FUNCTION "GestConsensoReal" : Void
{ S7_Optimized_Access := 'TRUE' }
VERSION : 0.1
   VAR_INPUT
      K_SegnaleMacchina : Int;
      K_Consenso : Int;
      K_TipoSendReceive : Int;   // Indica se è un segnale send o recive
      SegnaleIn : Real;   // Segnale in ingresso al blocco da inviare o ricevuto
   END_VAR

   VAR_OUTPUT
      OutSegnale : Real;
   END_VAR

   VAR_TEMP
      SegnaleForzatoOn : Bool;
      SegnaleForzatoOff : Bool;
      AbilitaTimeoutForzature : Bool;
      TimeoutForzature : Bool;
      ResettaForzature : Bool;
      PreOutSegnale : Real;
      StatoHmi : Int;
   END_VAR


BEGIN
	REGION Gestione delle forzature ad Hmi
	    #SegnaleForzatoOn := "SegnaliMacchina".S[#K_SegnaleMacchina].SR[#K_TipoSendReceive]."Real"[#K_Consenso].Hmi.ForzaturaOn;
	    #SegnaleForzatoOff := "SegnaliMacchina".S[#K_SegnaleMacchina].SR[#K_TipoSendReceive]."Real"[#K_Consenso].Hmi.ForzaturaOff;
	    #AbilitaTimeoutForzature := "SegnaliMacchina".S[#K_SegnaleMacchina].SR[#K_TipoSendReceive]."Real"[#K_Consenso].Prm.AbilitaScadenzaForzatura;
	    #TimeoutForzature := "SegnaliMacchina".S[#K_SegnaleMacchina].SR[#K_TipoSendReceive]."Real"[#K_Consenso].Prm.TempoScadenzaForzatura.O;
	    #ResettaForzature := #TimeoutForzature OR (#SegnaleForzatoOn AND #SegnaleForzatoOff);
	    "T_ON"(I_CicloCPU := "Zona".Comuni.TempoCicloCpu_r,
	           I_StartConteggio := (#SegnaleForzatoOn OR #SegnaleForzatoOff) AND #AbilitaTimeoutForzature,
	           IO_DatiTimer := "SegnaliMacchina".S[#K_SegnaleMacchina].SR[#K_TipoSendReceive]."Real"[#K_Consenso].Prm.TempoScadenzaForzatura);
	    IF #ResettaForzature THEN
	        "SegnaliMacchina".S[#K_SegnaleMacchina].SR[#K_TipoSendReceive]."Real"[#K_Consenso].Hmi.ForzaturaOn :=
	        "SegnaliMacchina".S[#K_SegnaleMacchina].SR[#K_TipoSendReceive]."Real"[#K_Consenso].Hmi.ForzaturaOff := False;
	    END_IF;
	    IF #SegnaleForzatoOn THEN
	        #PreOutSegnale := "SegnaliMacchina".S[#K_SegnaleMacchina].SR[#K_TipoSendReceive]."Real"[#K_Consenso].Hmi.ForzaturaValore;
	    ELSIF #SegnaleForzatoOff THEN
	        #PreOutSegnale := 0.0;
	    ELSE
	        #PreOutSegnale := #SegnaleIn + "SegnaliMacchina".S[#K_SegnaleMacchina].SR[#K_TipoSendReceive]."Real"[#K_Consenso].In.Segnale;
	    END_IF;
	END_REGION ;
	REGION Stato Hmi
	    IF #SegnaleForzatoOn THEN
	        #StatoHmi := 2;
	    ELSIF #SegnaleForzatoOff THEN
	        #StatoHmi := 3;
	    ELSIF #PreOutSegnale <> 0.0 THEN
	        #StatoHmi := 1;
	        ELSE
	        #StatoHmi := 0;
	    END_IF;
	    "SegnaliMacchina".S[#K_SegnaleMacchina].SR[#K_TipoSendReceive]."Real"[#K_Consenso].Hmi.Stato := #StatoHmi;
	END_REGION ;
	REGION Uscita
	    #OutSegnale := "SegnaliMacchina".S[#K_SegnaleMacchina].SR[#K_TipoSendReceive]."Real"[#K_Consenso].Out.Segnale := #PreOutSegnale;
	    ENO := True;
	END_REGION ;
END_FUNCTION

